FUNCTION_BLOCK FB_SPR
VAR_INPUT
END_VAR
VAR_OUTPUT
END_VAR
VAR
	Pufferspeicher_Kaltwasser_195						: FB_PSp;
	Pufferspeicher_Warmwasser_295						: FB_PSp;
	Pufferspeicher_Heisswasser_395						: FB_PSp;
END_VAR

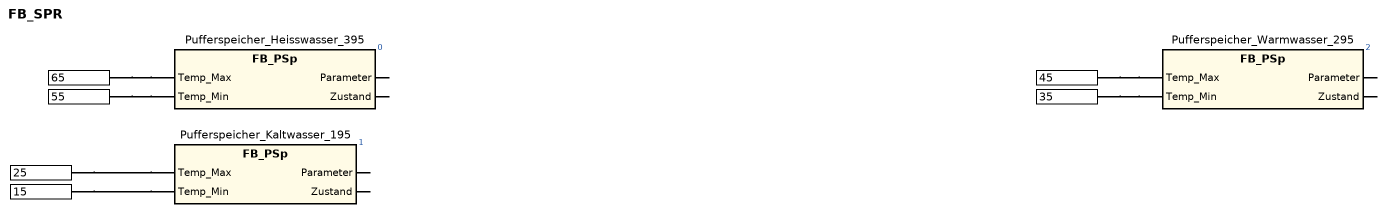
Pufferspeicher_Heisswasser_395(Temp_Max := 65, Temp_Min := 55); // FB_PSp
Pufferspeicher_Kaltwasser_195(Temp_Max := 25, Temp_Min := 15); // FB_PSp
Pufferspeicher_Warmwasser_295(Temp_Max := 45, Temp_Min := 35); // FB_PSp

END_FUNCTION_BLOCK

(* stored: Version 1.1.0.1, ProductVersion 3.1.4024.10
   POU FB_SPR: Id {533d91c1-442a-403a-a6ee-f4dbb832db78}, SpecialFunc None *)
